TYPE "bioPoT.DT"
TITLE = Batch I/O Polygon Table Data Type
// -- Woermann Automation --
AUTHOR : Woermann
VERSION : 0.1
	STRUCT
		Raw : ARRAY[0..15] of Real;	// (I) Input Values
		Val : ARRAY[0..15] of Real;	// (I) Output Values
	END_STRUCT;

END_TYPE

